// TIA Portal V16 export
// export: Created 2021-03-19T14:27:16.2808145Z, ExportSetting WithDefaults, DisplayName Totally Integrated Automation Portal, DisplayVersion V16 Update 3, DisplayName TIA Portal Version Control Interface, DisplayVersion V16 Update 2, DisplayName TIA Portal Openness, DisplayVersion V16 Update 3, DisplayName STEP 7 Professional, DisplayVersion V16 Update 3, DisplayName STEP 7 Safety, DisplayVersion V16, DisplayName WinCC Professional, DisplayVersion V16 Update 3
TYPE "UT02001_St_InstAnalogRead"
TITLE = Static UDT — Inst - Analogue Instrument Read and Scale
// Analogue Instrument Read and Scale
// stored: IsFailsafeCompliant false
   STRUCT
      revInfo { ExternalWritable := 'False'} : "UT01000_St_SysRevision";   // Revision information
      ___________0010_0 { ExternalAccessible := 'False'; ExternalVisible := 'False'; ExternalWritable := 'False'} : Int;
      ___________0010_1 { ExternalAccessible := 'False'; ExternalVisible := 'False'; ExternalWritable := 'False'} : Int;   // ▀▀▀▀ INSTRUMENT CONFIGURATION
      CONFIG_ALM_H_ENABLE { ExternalWritable := 'False'; S7_SetPoint := 'True'} : Bool;   // CONFIG — High alarm is enabled (1 = enabled, 0 = no alarm)
      CONFIG_ALM_L_ENABLE { ExternalWritable := 'False'; S7_SetPoint := 'True'} : Bool;   // CONFIG — Low alarm is enabled (1 = enabled, 0 = no alarm)
      CONFIG_WRN_H_ENABLE { ExternalWritable := 'False'; S7_SetPoint := 'True'} : Bool;   // CONFIG — High warning is enabled (1 = enabled, 0 = no warning)
      CONFIG_WRN_L_ENABLE { ExternalWritable := 'False'; S7_SetPoint := 'True'} : Bool;   // CONFIG — Low warning is enabled (1 = enabled, 0 = no warning)
      CONFIG_FP_DISABLE { ExternalWritable := 'False'; S7_SetPoint := 'True'} : Bool;   // CONFIG — Faceplate is disabled (1 = no Faceplate, 0 = normal)
      CONFIG_SIM_DISABLE { ExternalWritable := 'False'; S7_SetPoint := 'True'} : Bool;   // CONFIG — Simulation is disabled (1 = no Simulation, 0 = normal)
      CONFIG_RL_ENABLE { ExternalWritable := 'False'; S7_SetPoint := 'True'} : Bool;   // CONFIG — Remote/local mode enabled (1 = remote/local permitted, 0 = remote/local N/A)
      ___________0020_0 { ExternalAccessible := 'False'; ExternalVisible := 'False'; ExternalWritable := 'False'} : Int;
      ___________0020_1 { ExternalAccessible := 'False'; ExternalVisible := 'False'; ExternalWritable := 'False'} : Int;   // ▀▀▀▀ INSTRUMENT RANGE & SCALING DATA
      RANGE_RAW_MIN { ExternalWritable := 'False'; S7_SetPoint := 'True'} : Int;   // RANGE — Minimum value of the raw analogue signal (at the card)
      RANGE_RAW_MAX { ExternalWritable := 'False'; S7_SetPoint := 'True'} : Int;   // RANGE — Maximum value of the raw analogue signal (at the card)
      RANGE_SCALE_MIN { ExternalWritable := 'False'; S7_SetPoint := 'True'} : Real;   // RANGE — Minimum value of the scaled analogue signal [engineering units]
      RANGE_SCALE_MAX { ExternalWritable := 'False'; S7_SetPoint := 'True'} : Real;   // RANGE — Maximum value of the scaled analogue signal [engineering units]
      RANGE_OOR_PERCENT { ExternalWritable := 'False'; S7_SetPoint := 'True'} : Real;   // RANGE — Out of range percentage (of raw range), beyond which the instrument is out of range
      ___________0030_0 { ExternalAccessible := 'False'; ExternalVisible := 'False'; ExternalWritable := 'False'} : Int;
      ___________0030_1 { ExternalAccessible := 'False'; ExternalVisible := 'False'; ExternalWritable := 'False'} : Int;   // ▀▀▀▀ INSTRUMENT INFORMATION (TAG & UNITS)
      INFO_TAG { ExternalWritable := 'False'; S7_SetPoint := 'True'} : String[20];   // INFORMATION — Instrument ID tag
      INFO_UNITS { ExternalWritable := 'False'; S7_SetPoint := 'True'} : String[10];   // INFORMATION — Engineering units of the instrument (unit of measure)
      ___________0040_0 { ExternalAccessible := 'False'; ExternalVisible := 'False'; ExternalWritable := 'False'} : Int;
      ___________0040_1 { ExternalAccessible := 'False'; ExternalVisible := 'False'; ExternalWritable := 'False'} : Int;   // ▀▀▀▀ INSTRUMENT ALARM/WARNING & HYSTERESIS SETPOINTS
      SP_ALM_H_VAL { ExternalWritable := 'False'; S7_SetPoint := 'True'} : Real;   // SETPOINT — High alarm threshold value [engineering units]
      SP_ALM_L_VAL { ExternalWritable := 'False'; S7_SetPoint := 'True'} : Real;   // SETPOINT — Low alarm threshold value [engineering units]
      SP_WRN_H_VAL { ExternalWritable := 'False'; S7_SetPoint := 'True'} : Real;   // SETPOINT — High warning threshold value [engineering units]
      SP_WRN_L_VAL { ExternalWritable := 'False'; S7_SetPoint := 'True'} : Real;   // SETPOINT — Low warning threshold value [engineering units]
      SP_ALM_H_HYST_VAL { ExternalWritable := 'False'; S7_SetPoint := 'True'} : Real;   // SETPOINT — High alarm hysteresis value [engineering units]
      SP_ALM_L_HYST_VAL { ExternalWritable := 'False'; S7_SetPoint := 'True'} : Real;   // SETPOINT — Low alarm hysteresis value [engineering units]
      SP_WRN_H_HYST_VAL { ExternalWritable := 'False'; S7_SetPoint := 'True'} : Real;   // SETPOINT — High warning hysteresis value [engineering units]
      SP_WRN_L_HYST_VAL { ExternalWritable := 'False'; S7_SetPoint := 'True'} : Real;   // SETPOINT — Low warning hysteresis value [engineering units]
      ___________0050_0 { ExternalAccessible := 'False'; ExternalVisible := 'False'; ExternalWritable := 'False'} : Int;
      ___________0050_1 { ExternalAccessible := 'False'; ExternalVisible := 'False'; ExternalWritable := 'False'} : Int;   // ▀▀▀▀ INSTRUMENT TIMER DEFAULT VALUES
      TIME_ALM_H_ON_DEL { ExternalWritable := 'False'; S7_SetPoint := 'True'} : Real;   // TIMER — High alarm on delay time (activation delay), [seconds]
      TIME_ALM_L_ON_DEL { ExternalWritable := 'False'; S7_SetPoint := 'True'} : Real;   // TIMER — Low alarm on delay time (activation delay), [seconds]
      TIME_WRN_H_ON_DEL { ExternalWritable := 'False'; S7_SetPoint := 'True'} : Real;   // TIMER — High warning on delay time (activation delay), [seconds]
      TIME_WRN_L_ON_DEL { ExternalWritable := 'False'; S7_SetPoint := 'True'} : Real;   // TIMER — Low warning on delay time (activation delay), [seconds]
      TIME_ALM_H_OFF_DEL { ExternalWritable := 'False'; S7_SetPoint := 'True'} : Real;   // TIMER — High alarm off delay time (deactivation delay), [seconds]
      TIME_ALM_L_OFF_DEL { ExternalWritable := 'False'; S7_SetPoint := 'True'} : Real;   // TIMER — Low alarm off delay time (deactivation delay), [seconds]
      TIME_WRN_H_OFF_DEL { ExternalWritable := 'False'; S7_SetPoint := 'True'} : Real;   // TIMER — High warning off delay time (deactivation delay), [seconds]
      TIME_WRN_L_OFF_DEL { ExternalWritable := 'False'; S7_SetPoint := 'True'} : Real;   // TIMER — Low warning off delay time (deactivation delay), [seconds]
   END_STRUCT;
   // revInfo.REV_BLOCK := 'UT02001';
   // revInfo.REV_NUMBER := '001.000';
   // revInfo.REV_DATE := '2021-02-18';
   // revInfo.REV_AUTHOR := 'M. Gledhill ';
END_TYPE
